INTERFACE I_HaveProperties EXTENDS __SYSTEM.IQueryInterface

METHOD AddProperty
VAR_INPUT
	PropertyToAdd : I_Property;
END_VAR
END_METHOD

METHOD PUBLIC GetProperties : I_PropertyCollection
VAR_INPUT
END_VAR
END_METHOD

METHOD PUBLIC TryGetPropertyByName : BOOL
VAR_INPUT
	Name : T_MAXSTRING;
	Destination : REFERENCE TO I_Property;
END_VAR
END_METHOD

END_INTERFACE

(* stored: Version 1.1.0.1, ProductVersion 3.1.4024.12
   Itf I_HaveProperties: Id {c5806033-3adc-0f99-304c-e569fa5b2b9f}
   Method AddProperty: Id {629b0de3-c6af-0abc-2e2a-6709cf7d0165}
   Method GetProperties: Id {83aea430-01cb-0969-3ea6-7616f2695ec6}
   Method TryGetPropertyByName: Id {54f7a4bd-70df-0013-2d50-559760c48b28} *)
